FUNCTION_BLOCK FB_PersistentDataStorage IMPLEMENTS I_PersistentDataStorage
VAR_INPUT
END_VAR
VAR_OUTPUT
END_VAR
VAR
END_VAR

{warning 'Add property implementation'}
PROPERTY TriggerWriteOfPersistentData : BOOL
GET
END_GET
SET
END_SET
END_PROPERTY

END_FUNCTION_BLOCK

(* stored: Version 1.1.0.1
   POU FB_PersistentDataStorage: Id {63988f08-d855-49b0-a6b0-788913d53331}, SpecialFunc None
   Property TriggerWriteOfPersistentData: Id {92bcabd5-d918-4bec-962a-83f7bf4150cd}
   Get Get: Id {bac70043-b4e1-49f7-a385-1e9c35e95d0d}
   Set Set: Id {f3e4f96b-fd62-45d3-a29d-2b3ce53888ad} *)
